// TIA Portal V18 export
DATA_BLOCK "DB_MES_Monitoring"   // DB8
{ S7_Optimized_Access := 'TRUE' }
AUTHOR : caisik - mr. machinist
// stored: MemoryReserve 100
   VAR
      Diag { S7_SetPoint := 'True'} : "UDT_MES_Monitoring";
   END_VAR
BEGIN
END_DATA_BLOCK
